PROGRAM MAIN
VAR
	//Numbered variables for temperature and state
	nTankTemp :REAL := 25.0; 
	nState :INT := 10;
	
	//BOOL and Timer variables here
	bHeaterON :BOOL := FALSE;
	tSensorTimer :TON;
	IN: INT;
	PT: INT;
END_VAR

//Sensor made to set a timer on the loop to loop once every second.
tSensorTimer(IN:= NOT tSensorTimer.Q, PT:= T#1S);

//Introduction of a case state that has a different outcome for every integer
CASE nState OF
	10: //This is the start-up state
		bHeaterON := FALSE;
		IF nTankTemp < 40.0 THEN
			nState := 20;
			ELSE
				nState := 30;
		END_IF;
	20: //This is the heating-up state
		bHeaterON := TRUE;
		
		// Natural heating process limited by timer
		IF tSensorTimer.Q THEN
			nTankTemp := nTankTemp + 0.5;
		END_IF;
		
		//Detector to see if heat reaches a certain level
		IF nTankTemp > 60.0 THEN
			nState := 30;
		END_IF;
	
	30: //Cooling State
		bHeaterON := FALSE;
		
		//Natural process
		IF tSensorTimer.Q THEN
			nTankTemp := nTankTemp - 1;
		END_IF;
		
		//Sensor to switch state if temperature gets too low
		IF nTankTemp < 40.0 THEN
			nState := 20;
		END_IF;
END_CASE

END_PROGRAM

(* stored: Version 1.1.0.1, ProductVersion 3.1.4024.16
   POU MAIN: Id {bf6dad08-16ad-4349-8180-27d77fd387e0}, SpecialFunc None *)
